(* CoDeSys 2.3 export: ATRIBUTOS.EXP *)

(* Data type *)
TYPE Atributos :
STRUCT
	Fin_Operacion               : BOOL;
	Cond_Ini                         : BOOL;
	Estado_Emergencia    : BOOL;
END_STRUCT
END_TYPE
